FUNCTION_BLOCK FB_Axilon_Cooling_2f1p EXTENDS FB_Axilon_Cooling_1f1p
// Mirrors with 2 Cooling Flow Meters and 1 Pressure Meter
VAR_INPUT
END_VAR
VAR_OUTPUT
    {attribute 'pytmc' := '
        pv: FWM:2
        field: EGU lpm
        field: HIGH 2.3
        field: HIHI 3.0
        field: LOW 1.7
        field: LOLO 1.5
        io: i
    '}
    fFlow_2_val : LREAL;
END_VAR
VAR
    fbFlow_2 : FB_AnalogInput;
END_VAR

fbFlow_2(iTermBits:=15, fTermMax:=5.0427, fTermMin:=0.050472);
fFlow_2_val := fbFlow_2.fReal;

SUPER^();

END_FUNCTION_BLOCK

(* stored: Version 1.1.0.1, ProductVersion 3.1.4024.12
   POU FB_Axilon_Cooling_2f1p: Id {3668b105-d0a3-4fbc-a51d-7559f1a05e14}, SpecialFunc None *)
